KUKA KRL program: chk_w6_grp4_opn.src

&ACCESS RVO1
&REL 3
&COMMENT Check GRP ACCELO Z3 OPEN
DEF chk_w6_grp4_opn( )

; Check gripper accelo OPEN Z3.1/2/3/4/5
;//---- Start User-------

$TIMER[10] = 0
$TIMER_STOP[10] = FALSE

;FOLD WAIT FOR ( IN 60 'Z4 - Grampo Avancado - Accelo Bolha' );%{PE}%R 8.2.20,%MKUKATPBASIS,%CEXT_WAIT_FOR,%VEXT_WAIT_FOR,%P 2:, 4:, 5:$IN, 6:60, 7:Z4 - Grampo Avancado - Accelo Bolha, 9:
WAIT FOR  ( $IN[60] )
;ENDFOLD
;FOLD WAIT FOR ( NOT IN 59 'Z4 - Grampo Recuado - Accelo Bolha' );%{PE}%R 8.2.20,%MKUKATPBASIS,%CEXT_WAIT_FOR,%VEXT_WAIT_FOR,%P 2:, 4:NOT, 5:$IN, 6:59, 7:Z4 - Grampo Recuado - Accelo Bolha, 9:
WAIT FOR  (  NOT $IN[59] )
;ENDFOLD

$TIMER_STOP[10] = TRUE
$TIMER[10] = 0


;//---- End User---------

END
